{attribute 'OPC.UA.DA' := '0'}
TYPE HSPowermeter :
STRUCT
	PolarisationConfig : PolarisationConfig;
	RFactorSettings : RFactorSettings;
	ResponsivityConfig : ResponsivityConfig;
END_STRUCT
END_TYPE

(* stored: Version 1.1.0.1, ProductVersion 3.1.4024.10
   DUT HSPowermeter: Id {816dd29e-c99a-4fc3-8d76-ff6a5d75c779} *)
